{attribute 'analysis' := '-33'}
FUNCTION_BLOCK FB_L2SI_Flowmeter
VAR
    {attribute 'pytmc' := '
        pv: MA
        io: input
    '}
    fRaw AT %I*: INT;

    {attribute 'pytmc' := '
        pv: FLOW
        io: input
    '}
    fFlowRate: LREAL;
END_VAR

END_FUNCTION_BLOCK

(* stored: Version 1.1.0.1
   POU FB_L2SI_Flowmeter: Id {f4fe6025-68b2-43d4-8493-5a0f33999a1a}, SpecialFunc None *)
